FUNCTION_BLOCK MOTOR_DRIVER_SIMPLE (* Extracted Composite Function Block Type *)
  (* Standard: 61499-2 *)
  (* Version 4/28/2023, Dmitrii *)
  PACKAGE UAO.Hackathon;
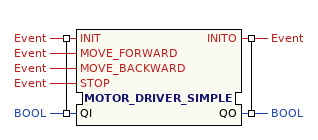
  EVENT_INPUT
    INIT WITH QI; (* Initializes the symbolic link data source FB with N (1 <= N <= 16) variables *)
    MOVE_FORWARD; (* Set Event *)
    MOVE_BACKWARD; (* Set Event *)
    STOP; (* Set Event *)
  END_EVENT
  EVENT_OUTPUT
    INITO WITH QO; (* Initialization confirm *)
  END_EVENT
  VAR_INPUT
    QI : BOOL; (* INIT event input qualifier *)
  END_VAR
  VAR_OUTPUT
    QO : BOOL; (* Output event qualifier *)
  END_VAR
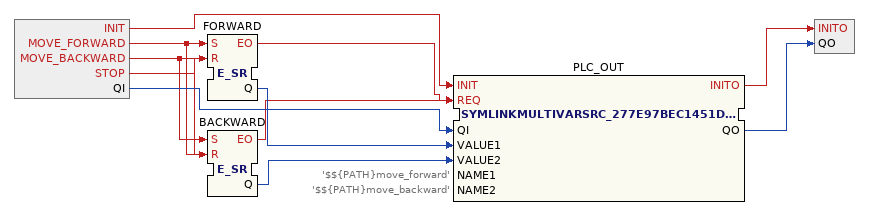
  FBS
    PLC_OUT : SYMLINKMULTIVARSRC_277E97BEC1451D2C(NAME1 := '$${PATH}move_forward', NAME2 := '$${PATH}move_backward'); {SET_ATTRIBUTE(Configuration.GenericFBType.InterfaceParams, Runtime.System#I:=2;VALUE${I$}:BOOL,BOOL)}
    FORWARD : E_SR;
    BACKWARD : E_SR;
  END_FBS
  EVENT_CONNECTIONS
    INIT TO PLC_OUT.INIT;
    PLC_OUT.INITO TO INITO;
    BACKWARD.EO TO PLC_OUT.REQ;
    FORWARD.EO TO PLC_OUT.REQ;
    MOVE_FORWARD TO FORWARD.S;
    MOVE_BACKWARD TO BACKWARD.S;
    MOVE_FORWARD TO BACKWARD.R;
    MOVE_BACKWARD TO FORWARD.R;
    STOP TO FORWARD.R;
    STOP TO BACKWARD.R;
  END_CONNECTIONS
  DATA_CONNECTIONS
    QI TO PLC_OUT.QI;
    PLC_OUT.QO TO QO;
    FORWARD.Q TO PLC_OUT.VALUE1;
    BACKWARD.Q TO PLC_OUT.VALUE2;
  END_CONNECTIONS
END_FUNCTION_BLOCK
